(* IEC 61131-3 sources: programs/VI-54/VI-54_20171205/VI-54_20171205/Stations/PLC_VI54/VI-54_171014/Class/ProductTriggerPositions, 1 file *)

(* ---- ProductTriggerPositions.st ---- *)
(*!
<Class
	Name               = "ProductTriggerPositions"
	Revision           = "0.0"
	RealtimeTask       = "true"
	CyclicTask         = "false"
	BackgroundTask     = "false"
	Sigmatek           = "false"
	OSInterface        = "false"
	HighPriority       = "false"
	Automatic          = "false"
	UpdateMode         = "Prescan"
	SharedCommandTable = "true"
	Objectsize         = "(870,120)">
	<Channels>
		<Server Name="__________" Visualized="false" Initialize="false" WriteProtected="true" Retentive="false"/>
		<Server Name="___________" Visualized="false" Initialize="false" WriteProtected="true" Retentive="false"/>
		<Server Name="ActProdPos" Visualized="true" Initialize="false" WriteProtected="true" Retentive="false"/>
		<Server Name="Comm" Visualized="true" Initialize="false" WriteProtected="true" Retentive="false"/>
		<Server Name="inpProductCntr" Visualized="true" Initialize="false" WriteProtected="true" Retentive="false" Comment="When the sensor is triggerd, the inpProductCntr will rise"/>
		<Server Name="MaxProdCntr" Visualized="false" Initialize="false" WriteProtected="true" Retentive="false"/>
		<Server Name="NewLookingBeltPos" Visualized="true" Initialize="false" WriteProtected="true" Retentive="false"/>
		<Server Name="outProductCntr" Visualized="true" Initialize="false" WriteProtected="true" Retentive="false" Comment="When the TriggerOffset is gone, the outProductCntr will rise"/>
		<Server Name="OutputTrigger" Visualized="true" Initialize="false" WriteProtected="true" Retentive="false"/>
		<Server Name="OutputTriggerTime" Visualized="true" Initialize="true" WriteProtected="false" Retentive="File"/>
		<Server Name="TriggerOffset" Visualized="true" Initialize="false" WriteProtected="true" Retentive="false"/>
		<Client Name="EncPos" Required="true" Internal="false"/>
		<Client Name="inpCntr" Required="false" Internal="false"/>
		<Client Name="iTrigger" Required="true" Internal="false"/>
		<Client Name="Motion" Required="true" Internal="false"/>
		<Client Name="Standard1" Required="true" Internal="true"/>
	</Channels>
	<Network Name="ProductTriggerPositions">
		<!-- List of Components in this network -->
		<Components>
			<Object
				Name           = "Standard1"
				Class          = "Standard"
				Position       = "(270,270)"
				Visualized     = "false"
				BackgroundTime = "1000 ms">
				<Channels>
					<Server Name="ClassSvr"/>
				</Channels>
			</Object>
		</Components>
		<Comments>
		</Comments>
		<!-- List of Connections in this network -->
		<Connections>
			<Connection Source="this.Standard1" Destination="Standard1.ClassSvr"/>
		</Connections>
		<!-- Headerfiles -->
		<Options>
		</Options>
	</Network>
</Class>
*)
ProductTriggerPositions : CLASS
	TYPE
#pragma pack(push, 1)
	  OutInfoStr : STRUCT  //! <Type Public="true" Name="OutInfoStr"/>
	    TriggerState : DINT;
	    PositionState : DINT;
	  END_STRUCT;
#pragma pack(pop)
#pragma pack(push, 1)
	  TriggerInfoStr : STRUCT  //! <Type Public="true" Name="TriggerInfoStr"/>
	    iFcBeltPos : DINT;
	    iOffsetBeltPos : DINT;
	    ProdNbr : DINT;
	    ProdGescand : DINT;
	    ProdPos : DINT;
	  END_STRUCT;
#pragma pack(pop)
	END_TYPE
  //Servers:
	Comm 	: SvrChCmd_DINT;
	__________ 	: SvrCh_DINT;
	TriggerOffset 	: SvrCh_DINT;
	NewLookingBeltPos 	: SvrCh_DINT;
	inpProductCntr 	: SvrCh_UDINT;
	outProductCntr 	: SvrCh_UDINT;
	MaxProdCntr 	: SvrCh_DINT;
	___________ 	: SvrCh_DINT;
	OutputTrigger 	: SvrCh_DINT;
	ActProdPos 	: SvrCh_DINT;
	OutputTriggerTime 	: SvrCh_DINT;
  //Clients:
	Motion 	: CltChCmd__LMCAxis;
	EncPos 	: CltCh_DINT;
	iTrigger 	: CltChCmd_PositionFilterIFC;
	inpCntr 	: CltCh_DINT;
	Standard1 	: CltChCmd_Standard;
  //Variables:
		TriggerInformation : ARRAY [0..255] OF TriggerInfoStr;

		Cntr 	: USINT;
		ReadCntr 	: USINT;
		IntUnits 	: DINT;
		ExtUnits 	: DINT;
		rMulDiv 	: REAL;
		DeltaOffset 	: REAL;
		DeltaOffsetMM 	: DINT;
		NumberOfProduct 	: DINT;
		ActProdNumber 	: DINT;
		TriggerInfo 	: TriggerStr;
  //Functions:

	FUNCTION VIRTUAL GLOBAL RtWork
		VAR_INPUT
			EAX 	: UDINT;
		END_VAR
		VAR_OUTPUT
			state (EAX) 	: UDINT;
		END_VAR;

	FUNCTION GLOBAL InputTrigger
		VAR_OUTPUT
			State 	: DINT;
		END_VAR;

	FUNCTION GLOBAL OffsetTrigger
		VAR_OUTPUT
			State 	: OutInfoStr;
		END_VAR;

	FUNCTION GLOBAL SetTriggerOffset
		VAR_INPUT
			State 	: DINT;
		END_VAR;

	FUNCTION GLOBAL SetTriggerArray;

	FUNCTION GLOBAL ReadTriggerArray;

	FUNCTION GLOBAL SetMaxProducts
		VAR_INPUT
			Amount 	: DINT;
		END_VAR;

	FUNCTION GLOBAL ProdNbr
		VAR_OUTPUT
			Nbr 	: DINT;
		END_VAR;
  //Tables:
	FUNCTION @STD
		VAR_OUTPUT
			ret_code	: CONFSTATES;
		END_VAR;
	FUNCTION GLOBAL TAB @CT_;
END_CLASS;

#pragma using Standard
#pragma usingLtd _LMCAxis
#pragma usingLtd PositionFilterIFC

FUNCTION VIRTUAL GLOBAL ProductTriggerPositions::RtWork
	VAR_INPUT
		EAX 	: UDINT;
	END_VAR
	VAR_OUTPUT
		state (EAX) 	: UDINT;
	END_VAR

  // Read inputs
  Motion      := Motion.Read();
  EncPos      := EncPos.Read();
  TriggerInfo := iTrigger.ReadTrigger();
  iTrigger    := TriggerInfo.TriggerState;

  // open methodes
  SetTriggerArray(); // Set the input fotocel into a register
  ReadTriggerArray();

  // Read axle variables
  IntUnits := Motion.ReadParameter(ParNr:=LMCAXIS_PAR_RD_INTUNITS, mode:=0);
  ExtUnits := Motion.ReadParameter(ParNr:=LMCAXIS_PAR_RD_EXTUNITS, mode:=0);
  rMulDiv  := to_real(IntUnits) / to_real(ExtUnits);

	state := READY;

END_FUNCTION

FUNCTION GLOBAL ProductTriggerPositions::SetTriggerArray

  // Scan rising edge of the trigger input
  if Standard1.R_TRIG(CLK:= iTrigger) = 1 then

      NumberOfProduct += 1;

      // Set information in Array
      TriggerInformation[Cntr].iFcBeltPos     := EncPos;
      TriggerInformation[Cntr].iOffsetBeltPos := TriggerOffset;
      TriggerInformation[Cntr].ProdNbr        := NumberOfProduct;
      TriggerInformation[Cntr].ProdGescand    := 1;
      TriggerInformation[Cntr].ProdPos        := to_dint(TriggerInfo.PositionState);

      Cntr += 1;
      inpProductCntr := to_udint Cntr;

      if NumberOfProduct >= MaxProdCntr then // because we start at '0'
        NumberOfProduct := 0;
      end_if;
  end_if;

END_FUNCTION

FUNCTION GLOBAL ProductTriggerPositions::ReadTriggerArray

  if ReadCntr <> Cntr then
    DeltaOffset   := to_real(EncPos - TriggerInformation[ReadCntr].iFcBeltPos);    //counts sinds foto
    DeltaOffsetMM := to_dint(to_real DeltaOffset * rMulDiv);
    if DeltaOffsetMM >= TriggerInformation[ReadCntr].iOffsetBeltPos then
      ActProdPos                                  := TriggerInformation[ReadCntr].ProdPos;
      ActProdNumber                               := TriggerInformation[ReadCntr].ProdNbr;
      TriggerInformation[ReadCntr].iFcBeltPos     := 0;
      TriggerInformation[ReadCntr].iOffsetBeltPos := 0;
      TriggerInformation[ReadCntr].ProdNbr        := 0;
      TriggerInformation[ReadCntr].ProdGescand    := 0;
      TriggerInformation[ReadCntr].ProdPos        := 0;

      ReadCntr += 1;
      outProductCntr := to_udint ReadCntr;
      OutputTrigger := 1;

    end_if;
  end_if;

  // Hold output trigger high for 50ms
  if OutputTriggerTime < 50 then
    OutputTriggerTime := 50;
  end_if;

  // Hold output trigger high for 50ms
  if Standard1.TON(IN:= OutputTrigger, PT:= OutputTriggerTime) then
    OutputTrigger := 0;
  end_if;

END_FUNCTION

FUNCTION GLOBAL ProductTriggerPositions::InputTrigger
	VAR_OUTPUT
		State 	: DINT;
	END_VAR

  State := iTrigger;

END_FUNCTION

FUNCTION GLOBAL ProductTriggerPositions::OffsetTrigger
	VAR_OUTPUT
		State 	: OutInfoStr;
	END_VAR

  State.TriggerState  := OutputTrigger;
  State.PositionState := ActProdPos;

END_FUNCTION

FUNCTION GLOBAL ProductTriggerPositions::ProdNbr
	VAR_OUTPUT
		Nbr 	: DINT;
	END_VAR

  Nbr := ActProdNumber;

END_FUNCTION

FUNCTION GLOBAL ProductTriggerPositions::SetTriggerOffset
	VAR_INPUT
		State 	: DINT;
	END_VAR

  TriggerOffset := State;

END_FUNCTION

FUNCTION GLOBAL ProductTriggerPositions::SetMaxProducts
	VAR_INPUT
		Amount 	: DINT;
	END_VAR

  MaxProdCntr := Amount;

END_FUNCTION
